SUPER^(); // FB_BA_View
Input(bVal := bVal); // FB_BA_BI
bPresentValue := Input.bPresentValue;

METHOD FB_init : BOOL
VAR_INPUT
	bInitRetains : BOOL; // if TRUE, the retain variables are initialized (warm start / cold start)
	bInCopyCode : BOOL;  // if TRUE, the instance afterwards gets moved into the copy code (online change)
END_VAR
Input.iParent						:= THIS^;
Input.iLabel						:= LblUniFieldDevice.SensorBinary_Input;	
Input.sObjectName					:= '{Idx=01}';	
Input.sDeviceType					:= '';
Input.bEnOutOfService				:= FALSE;
Input.sActiveText 					:= txtEvent_Triggered;
Input.sInactiveText 				:= txtEvent_Normal;
Input.nStateChangeCount				:= 0;
Input.nActiveTimeElapsed			:= 0;
Input.nEventClassID					:= EC_ID.NC30;
Input.stTimeDelay.nToNormal			:= BA2_Param.nDefTimeDelay_ToNormal;
Input.stTimeDelay.nToAbnormal		:= BA2_Param.nDefTimeDelay_ToAbnormal;
Input.bAlarmValue					:= TRUE;
Input.bAcknowledgeRm				:= FALSE;		
Input.aEventTransitionText[1]		:= txtEvent_Triggered;
Input.aEventTransitionText[2]		:= txtEvent_Error;
Input.aEventTransitionText[3]		:= txtEvent_Normal;
Input.bEventDetectionEnable			:= TRUE;
Input.aEventEnable[1]				:= TRUE;			//	to_offnormal
Input.aEventEnable[2]				:= TRUE;			//	to_fault
Input.aEventEnable[3]				:= TRUE;			//	to_normal
Input.eEnPlantLock					:= E_BA_LockPriority.eNoLock;
END_METHOD

END_FUNCTION_BLOCK

// ---- Templates/POUs/Universal/Sensor/FB_BA_SensorAnalog.TcPOU
{region '#Template'}
	{attribute 'Version' := '1.2.1.0'}
	{attribute 'Tags' := '"LCID": "1031", "Text": "Universal, Sensor, AI"'}
	{attribute 'Tags' := '"LCID": "1033", "Text": "Universal, Sensor, AI"'}
	{attribute 'Using' := '"Type": "Template", "URI": "EC_AMEV"'}
	{attribute 'Using' := '"Type": "Template", "URI": "BA2_Param"'}
	{attribute 'Description' := '"LCID": "1031", "Text": "AI ohne IO"'}
	{attribute 'Description' := '"LCID": "1033", "Text": "AI without IO"'}
{endregion}
FUNCTION_BLOCK FB_BA_SensorAnalog EXTENDS FB_BA_View
VAR_INPUT
	fVal					: REAL;
END_VAR
VAR_INPUT CONSTANT
	MV						: FB_BA_AI;		
END_VAR
VAR_OUTPUT
	fPresentValue			: REAL;
	bEvent					: BOOL;
	eEventState				: E_BA_EventState;	
END_VAR
VAR
END_VAR

SUPER^(); // FB_BA_View
MV(fVal := fVal); // FB_BA_AI
bEvent := MV.bEvent;
eEventState := MV.eEventState;
fPresentValue := MV.fPresentValue;

METHOD FB_init : BOOL
VAR_INPUT
	bInitRetains : BOOL; // if TRUE, the retain variables are initialized (warm start / cold start)
	bInCopyCode : BOOL;  // if TRUE, the instance afterwards gets moved into the copy code (online change)
END_VAR
MV.iParent						:= THIS^;		
MV.iLabel 						:= LblUniFieldDevice.SensorAnalog_MV;
MV.sObjectName					:= '{Idx=01}';
MV.sDeviceType					:= '';
MV.bEnOutOfService				:= FALSE;
MV.eUnit						:= E_BA_Unit.eTemperature_DegreesCelsius;
MV.fCOVIncrement				:= BA2_Param.fDefCOVIncrement;
MV.nEventClassID				:= EC_ID.NC30;
MV.stTimeDelay.nToNormal		:= BA2_Param.nDefTimeDelay_ToNormal;
MV.stTimeDelay.nToAbnormal		:= BA2_Param.nDefTimeDelay_ToAbnormal;
MV.stHighLimit.bEnable			:= FALSE;
MV.stHighLimit.fValue			:= 0.0;		
MV.stLowLimit.bEnable			:= FALSE;
MV.stLowLimit.fValue			:= 0.0;
MV.fLimitDeadband 				:= BA2_Param.fDefLimitDeadband;
MV.bAcknowledgeRm				:= FALSE;	
MV.aEventTransitionText[1]		:= txtEvent_Exceeded;
MV.aEventTransitionText[2]		:= txtEvent_Disturb;
MV.aEventTransitionText[3]		:= txtEvent_Normal;
MV.bEventDetectionEnable		:= TRUE;
MV.aEventEnable[1]				:= TRUE;			//	to_offnormal
MV.aEventEnable[2]				:= TRUE;			//	to_fault
MV.aEventEnable[3]				:= TRUE;			//	to_normal
MV.eEnPlantLock					:= E_BA_LockPriority.eNoLock;
END_METHOD

END_FUNCTION_BLOCK

// ---- Templates/POUs/Universal/Sensor/FB_BA_MeasuredValueCardinal.TcPOU
{region '#Template'}
	{attribute 'Version' := '1.2.1.0'}
	{attribute 'Tags' := '"LCID": "1031", "Text": "Universal, Sensor, AI"'}
	{attribute 'Tags' := '"LCID": "1033", "Text": "Universal, Sensor, AI"'}
	{attribute 'Using' := '"Type": "Template", "URI": "EC_AMEV"'}
	{attribute 'Using' := '"Type": "Template", "URI": "BA2_Param"'}
	{attribute 'Description' := '"LCID": "1031", "Text": "Kombination 4x AI ohne IO"'}
	{attribute 'Description' := '"LCID": "1033", "Text": "Combination 4x AI without IO"'}
{endregion}
FUNCTION_BLOCK FB_BA_MeasuredValueCardinal EXTENDS FB_BA_View
VAR_INPUT
	fVal_N					: REAL;
	fVal_S					: REAL;
	fVal_E					: REAL;
	fVal_W					: REAL;
END_VAR
VAR_INPUT CONSTANT
	MV_N					: FB_BA_AI;		
	MV_S					: FB_BA_AI;	
	MV_E					: FB_BA_AI;		
	MV_W					: FB_BA_AI;			
END_VAR
VAR_OUTPUT
	fPresentValueN			: REAL;
	fPresentValueS			: REAL;
	fPresentValueE			: REAL;
	fPresentValueW			: REAL;
END_VAR
VAR
END_VAR

SUPER^(); // FB_BA_View
MV_N(fVal := fVal_N); // FB_BA_AI
fPresentValueN := MV_N.fPresentValue;
MV_S(fVal := fVal_S); // FB_BA_AI
fPresentValueS := MV_S.fPresentValue;
MV_E(fVal := fVal_E); // FB_BA_AI
fPresentValueE := MV_E.fPresentValue;
MV_W(fVal := fVal_W); // FB_BA_AI
fPresentValueW := MV_W.fPresentValue;

METHOD FB_init : BOOL
VAR_INPUT
	bInitRetains : BOOL; // if TRUE, the retain variables are initialized (warm start / cold start)
	bInCopyCode : BOOL;  // if TRUE, the instance afterwards gets moved into the copy code (online change)
END_VAR
MV_N.iParent						:= THIS^;		
MV_N.iLabel 						:= LblUniFieldDevice.SensorAnalog_MV_N;
MV_N.sObjectName					:= '{Idx=01}';
MV_N.sDeviceType					:= '';
MV_N.bEnOutOfService				:= FALSE;
MV_N.eUnit							:= E_BA_Unit.eTemperature_DegreesCelsius;
MV_N.fCOVIncrement					:= BA2_Param.fDefCOVIncrement;
MV_N.nEventClassID					:= EC_ID.NC30;
MV_N.stTimeDelay.nToNormal			:= BA2_Param.nDefTimeDelay_ToNormal;
MV_N.stTimeDelay.nToAbnormal		:= BA2_Param.nDefTimeDelay_ToAbnormal;
MV_N.stHighLimit.bEnable			:= FALSE;
MV_N.stHighLimit.fValue				:= 0.0;		
MV_N.stLowLimit.bEnable				:= FALSE;
MV_N.stLowLimit.fValue				:= 0.0;
MV_N.fLimitDeadband 				:= BA2_Param.fDefLimitDeadband;
MV_N.bAcknowledgeRm					:= FALSE;	
MV_N.aEventTransitionText[1]		:= txtEvent_Exceeded;
MV_N.aEventTransitionText[2]		:= txtEvent_Disturb;
MV_N.aEventTransitionText[3]		:= txtEvent_Normal;
MV_N.bEventDetectionEnable			:= FALSE;
MV_N.aEventEnable[1]				:= TRUE;			//	to_offnormal
MV_N.aEventEnable[2]				:= TRUE;			//	to_fault
MV_N.aEventEnable[3]				:= TRUE;			//	to_normal
MV_N.eEnPlantLock					:= E_BA_LockPriority.eNoLock;			

MV_S.iParent						:= THIS^;		
MV_S.iLabel 						:= LblUniFieldDevice.SensorAnalog_MV_S;
MV_S.sObjectName					:= '{Idx=02}';
MV_S.sDeviceType					:= '';
MV_S.bEnOutOfService				:= FALSE;
MV_S.eUnit							:= E_BA_Unit.eTemperature_DegreesCelsius;
MV_S.fCOVIncrement					:= BA2_Param.fDefCOVIncrement;
MV_S.nEventClassID					:= EC_ID.NC30;
MV_S.stTimeDelay.nToNormal			:= BA2_Param.nDefTimeDelay_ToNormal;
MV_S.stTimeDelay.nToAbnormal		:= BA2_Param.nDefTimeDelay_ToAbnormal;
MV_S.stHighLimit.bEnable			:= FALSE;
MV_S.stHighLimit.fValue				:= 0.0;		
MV_S.stLowLimit.bEnable				:= FALSE;
MV_S.stLowLimit.fValue				:= 0.0;
MV_S.fLimitDeadband 				:= BA2_Param.fDefLimitDeadband;
MV_S.bAcknowledgeRm					:= FALSE;	
MV_S.aEventTransitionText[1]		:= txtEvent_Exceeded;
MV_S.aEventTransitionText[2]		:= txtEvent_Disturb;
MV_S.aEventTransitionText[3]		:= txtEvent_Normal;
MV_S.bEventDetectionEnable			:= FALSE;
MV_S.aEventEnable[1]				:= TRUE;			//	to_offnormal
MV_S.aEventEnable[2]				:= TRUE;			//	to_fault
MV_S.aEventEnable[3]				:= TRUE;			//	to_normal
MV_S.eEnPlantLock					:= E_BA_LockPriority.eNoLock;

MV_E.iParent						:= THIS^;		
MV_E.iLabel 						:= LblUniFieldDevice.SensorAnalog_MV_E;
MV_E.sObjectName					:= '{Idx=03}';
MV_E.sDeviceType					:= '';
MV_E.bEnOutOfService				:= FALSE;
MV_E.eUnit							:= E_BA_Unit.eTemperature_DegreesCelsius;
MV_E.fCOVIncrement					:= BA2_Param.fDefCOVIncrement;
MV_E.nEventClassID					:= EC_ID.NC30;
MV_E.stTimeDelay.nToNormal			:= BA2_Param.nDefTimeDelay_ToNormal;
MV_E.stTimeDelay.nToAbnormal		:= BA2_Param.nDefTimeDelay_ToAbnormal;
MV_E.stHighLimit.bEnable			:= FALSE;
MV_E.stHighLimit.fValue				:= 0.0;		
MV_E.stLowLimit.bEnable				:= FALSE;
MV_E.stLowLimit.fValue				:= 0.0;
MV_E.fLimitDeadband 				:= BA2_Param.fDefLimitDeadband;
MV_E.bAcknowledgeRm					:= FALSE;	
MV_E.aEventTransitionText[1]		:= txtEvent_Exceeded;
MV_E.aEventTransitionText[2]		:= txtEvent_Disturb;
MV_E.aEventTransitionText[3]		:= txtEvent_Normal;
MV_E.bEventDetectionEnable			:= FALSE;
MV_E.aEventEnable[1]				:= TRUE;			//	to_offnormal
MV_E.aEventEnable[2]				:= TRUE;			//	to_fault
MV_E.aEventEnable[3]				:= TRUE;			//	to_normal
MV_E.eEnPlantLock					:= E_BA_LockPriority.eNoLock;

MV_W.iParent						:= THIS^;		
MV_W.iLabel 						:= LblUniFieldDevice.SensorAnalog_MV_W;
MV_W.sObjectName					:= '{Idx=04}';
MV_W.sDeviceType					:= '';
MV_W.bEnOutOfService				:= FALSE;
MV_W.eUnit							:= E_BA_Unit.eTemperature_DegreesCelsius;
MV_W.fCOVIncrement					:= BA2_Param.fDefCOVIncrement;
MV_W.nEventClassID					:= EC_ID.NC30;
MV_W.stTimeDelay.nToNormal			:= BA2_Param.nDefTimeDelay_ToNormal;
MV_W.stTimeDelay.nToAbnormal		:= BA2_Param.nDefTimeDelay_ToAbnormal;
MV_W.stHighLimit.bEnable			:= FALSE;
MV_W.stHighLimit.fValue				:= 0.0;		
MV_W.stLowLimit.bEnable				:= FALSE;
MV_W.stLowLimit.fValue				:= 0.0;
MV_W.fLimitDeadband 				:= BA2_Param.fDefLimitDeadband;
MV_W.bAcknowledgeRm					:= FALSE;	
MV_W.aEventTransitionText[1]		:= txtEvent_Exceeded;
MV_W.aEventTransitionText[2]		:= txtEvent_Disturb;
MV_W.aEventTransitionText[3]		:= txtEvent_Normal;
MV_W.bEventDetectionEnable			:= FALSE;
MV_W.aEventEnable[1]				:= TRUE;			//	to_offnormal
MV_W.aEventEnable[2]				:= TRUE;			//	to_fault
MV_W.aEventEnable[3]				:= TRUE;			//	to_normal
MV_W.eEnPlantLock					:= E_BA_LockPriority.eNoLock;
END_METHOD

END_FUNCTION_BLOCK

// ---- Templates/POUs/Trade/AC/Setpoint/Temperature/FB_BA_AC_SpTRm_01.TcPOU
{region '#Template'}
	{attribute 'Version' := '1.0.0.0'}
	{attribute 'Tags' := '"LCID": "1031", "Text": "AC, Setpoint, Room temperature"'}
	{attribute 'Tags' := '"LCID": "1033", "Text": "AC, Setpoint, Room temperature"'}
	{attribute 'Description' := '"LCID": "1031", "Text": "Sollwert Raumtemperatur"'}
	{attribute 'Description' := '"LCID": "1033", "Text": "Setpoint room temperature"'}
{endregion}
FUNCTION_BLOCK FB_BA_AC_SpTRm_01 EXTENDS FB_BA_View
VAR_INPUT
	fTWth					: REAL;	
END_VAR
VAR_OUTPUT
	fSp						: REAL;
END_VAR
VAR_INPUT CONSTANT
	X1						: FB_BA_AV_Op;
	X2						: FB_BA_AV_Op;
	X3						: FB_BA_AV_Op;
	X4						: FB_BA_AV_Op;
	Y1						: FB_BA_AV_Op;
	Y2_3					: FB_BA_AV_Op;	
	Y4						: FB_BA_AV_Op;
	Sp						: FB_BA_AV_Op;						
END_VAR
VAR
	Scale					: FB_BA_Chrct04;	
END_VAR

SUPER^(); // FB_BA_View
X1(); // FB_BA_AV_Op
X2(); // FB_BA_AV_Op
X3(); // FB_BA_AV_Op
X4(); // FB_BA_AV_Op
Y1(); // FB_BA_AV_Op
Y2_3(); // FB_BA_AV_Op
Y4(); // FB_BA_AV_Op
Scale(
    fX := fTWth,
    fX01 := X1.fPresentValue,
    fX02 := X2.fPresentValue,
    fX03 := X3.fPresentValue,
    fX04 := X4.fPresentValue,
    fY01 := Y1.fPresentValue,
    fY02 := Y2_3.fPresentValue,
    fY03 := Y2_3.fPresentValue,
    fY04 := Y4.fPresentValue,
    fYMin := Y2_3.fPresentValue,
    fYMax := Y4.fPresentValue); // FB_BA_Chrct04
Sp(fValuePgm := Scale.fCalcVal); // FB_BA_AV_Op
fSp := Sp.fPresentValue;

METHOD FB_init : BOOL
VAR_INPUT
	bInitRetains : BOOL; // if TRUE, the retain variables are initialized (warm start / cold start)
	bInCopyCode : BOOL;  // if TRUE, the instance afterwards gets moved into the copy code (online change)
END_VAR
X1.iParent				:= THIS^;
X1.iLabel				:= LblCmpAC.SpTRm_X1;			
X1.sObjectName			:= '{Idx=01}';								 	 
X1.eUnit				:= E_BA_Unit.eTemperature_DegreesCelsius;  
X1.fValueRm				:= -15.0;
X1.fCOVIncrement		:= BA2_Param.fDefCOVIncrement;

X2.iParent				:= THIS^;
X2.iLabel				:= LblCmpAC.SpTRm_X2;			
X2.sObjectName			:= '{Idx=02}';	 	 
X2.eUnit				:= E_BA_Unit.eTemperature_DegreesCelsius;  
X2.fValueRm				:= -5.0;
X2.fCOVIncrement		:= BA2_Param.fDefCOVIncrement;

X3.iParent				:= THIS^;
X3.iLabel				:= LblCmpAC.SpTRm_X3;			
X3.sObjectName			:= '{Idx=03}';								 	 
X3.eUnit				:= E_BA_Unit.eTemperature_DegreesCelsius;  
X3.fValueRm				:= 26.0;
X3.fCOVIncrement		:= BA2_Param.fDefCOVIncrement;

X4.iParent				:= THIS^;
X4.iLabel				:= LblCmpAC.SpTRm_X4;			
X4.sObjectName			:= '{Idx=04}';								 	 
X4.eUnit				:= E_BA_Unit.eTemperature_DegreesCelsius;  
X4.fValueRm				:= 32.0;
X4.fCOVIncrement		:= BA2_Param.fDefCOVIncrement;

Y1.iParent				:= THIS^;
Y1.iLabel				:= LblCmpAC.SpTRm_Y1;			
Y1.sObjectName			:= '{Idx=01}';								 	 
Y1.eUnit				:= E_BA_Unit.eTemperature_DegreesCelsius;  
Y1.fValueRm				:= 23.0;
Y1.fCOVIncrement		:= BA2_Param.fDefCOVIncrement;

Y2_3.iParent			:= THIS^;
Y2_3.iLabel				:= LblCmpAC.SpTRm_Y2_3;			
Y2_3.sObjectName		:= '{Idx=02}';								 	 
Y2_3.eUnit				:= E_BA_Unit.eTemperature_DegreesCelsius;  
Y2_3.fValueRm			:= 21.0;
Y2_3.fCOVIncrement		:= BA2_Param.fDefCOVIncrement;
	
Y4.iParent				:= THIS^;
Y4.iLabel				:= LblCmpAC.SpTRm_Y4;			
Y4.sObjectName			:= '{Idx=04}';								 	 
Y4.eUnit				:= E_BA_Unit.eTemperature_DegreesCelsius;  
Y4.fValueRm				:= 28.0;
Y4.fCOVIncrement		:= BA2_Param.fDefCOVIncrement;

Sp.iParent				:= THIS^;
Sp.iLabel				:= LblCmpAC.SpTRm_Sp;			
Sp.sObjectName			:= '{Idx=01}';								 	 
Sp.eUnit				:= E_BA_Unit.eTemperature_DegreesCelsius;
Sp.fCOVIncrement		:= BA2_Param.fDefCOVIncrement;
END_METHOD

END_FUNCTION_BLOCK
